{attribute 'linkalways'} 
{attribute 'no_explicit_call' := 'This FB is a CLASS and must be accessed using methods or properties'}
{attribute 'enable_dynamic_creation'}
FUNCTION_BLOCK FINAL LT_BYTE EXTENDS Node
VAR
	in1 : _BYTE(0);
	in2 : _BYTE(0);
	out : _BOOL(FALSE);
END_VAR

METHOD PUBLIC Clone : I_Node
VAR
	pNode : POINTER TO LT_BYTE;
END_VAR
pNode := __NEW(LT_BYTE);
Clone := pNode^;
END_METHOD

METHOD FB_init : BOOL
VAR_INPUT
	bInitRetains : BOOL; // if TRUE, the retain variables are initialized (warm start / cold start)
	bInCopyCode : BOOL;  // if TRUE, the instance afterwards gets moved into the copy code (online change)
END_VAR
AddInput('in1',THIS^.in1);
AddInput('in2',THIS^.in2);
AddOutput('out', THIS^.out);
END_METHOD

METHOD PROTECTED OnExecute
VAR
END_VAR
out.Value := in1.Value < in2.Value;
END_METHOD

END_FUNCTION_BLOCK

(* stored: Version 1.1.0.1, ProductVersion 3.1.4024.15
   POU LT_BYTE: Id {ef4a0234-bb8d-4b9b-821a-76858e04e4fa}, SpecialFunc None
   Folder Constructor: Id {ac4655f2-86f6-42e3-a3dd-73f68e57637e}
   Method Clone: Id {1b102ba2-3fc1-4e1a-b499-af14de1cf4a9}
   Method FB_init: Id {df80bd5c-fdbe-4066-8d00-45346ec3cb3a}
   Method OnExecute: Id {a5a70769-fd6c-4ed4-a065-c80f4da8d051} *)
